Staubli VAL3: getSize.pgx

public program getSize(num& x_nSize[])
begin
  // how many items
  call out:getSize(x_nSize)
end
